(*
:Author: 

	Takashi Ichihashi Beckhoff Automation co. ltd.
	
:Date:

	2023-03-09
	
Overview
==================



Infosys Link:  `https://infosys.beckhoff.com/content/1033/tf6420_tc3_database_server/8117583755.html?id=5199556541044360835 <https://infosys.beckhoff.com/content/1033/tf6420_tc3_database_server/8117583755.html?id=5199556541044360835>`

Quick start
======================

As first you have to deine data model that the sampling data to insert to influxDB measurement.  The data models are structured by parent and child that is corresponding data tags and fields on influxDB.

.. code:: DataTag structure

	TYPE DataTag:
	STRUCT
		{attribute 'TagName' := 'machine_id'}
		machine_id : STRING(255); // 設備名
		{attribute 'TagName' := 'data_type_id'}
		data_type_id : STRING(255); // 発生イベント種別
	END_STRUCT
	END_TYPE	

	
.. code:: DataField structure

	TYPE PerformanceData EXTENDS DataTag:
	STRUCT
		{attribute 'FieldName' := 'plc_task_time'}
		task_time: UDINT;
		{attribute 'FieldName' := 'cpu_usage'}
		cpu_usage: UDINT;
		{attribute 'FieldName' := 'latency'}
		latency: UDINT;
		{attribute 'FieldName' := 'max_latency'}
		max_latency: UDINT;
		{attribute 'FieldName' := 'exceed_counter'}
		exceed_counter: UDINT;
		{attribute 'FieldName' := 'ec_lost_frames'}
		ec_lost_frames: UDINT;
		{attribute 'FieldName' := 'ec_frame_rate'}
		ec_frame_rate: LREAL;
		{attribute 'FieldName' := 'ec_lost_q_frame'}
		ec_lost_q_frames: UDINT;
		{attribute 'FieldName' := 'ec_q_frame_rate'}
		ec_q_frame_rate: LREAL;
		{attribute 'FieldName' := 'executing'}
		executing: BOOL;
		{attribute 'FieldName' := 'DB_queue_count'}
		db_insert_queue_count: UDINT;
		{attribute 'FieldName' := 'DB_buffer_current_index'}
		current_index: UDINT;
		{attribute 'FieldName' := 'DB_buffer_next_index'}
		next_index: UDINT;
	
	END_STRUCT
	END_TYPE
	
*)

FUNCTION_BLOCK RecordSQL IMPLEMENTS IRecordDB
VAR_INPUT
	nDBID						: UDINT;					// Database ID for TF6420
	DB_Parameter				: Tc2_Utilities.T_Arg;
END_VAR
VAR_OUTPUT
	bBusy			: BOOL;	// In writing database
	bError			: BOOL; // Somthing wrong situation happend
	TcResult		: Tc3_Database.I_TcMessage; // Response message
    sErrorMessage	: STRING(255);	// Error message
END_VAR
VAR
	
	//for generating timestamp
	fbGetSystemTime1: GetSystemTime;
	dwTimeLoDW: DWORD;
	dwTimeHiDW: DWORD;
	tFileTime: T_FILETIME;
	nTimestamp: LINT;
	
	//for insert samples
	fbPLCDBCmd: FB_PLCDBCmdEvt(sNetID := '', tTimeout := T#19S);
	_query								: STRING(512);
	
	// Variables for queue feature
	get_data_t 			: T_Arg;
	get_data 			: DbInsertCommand;
	State				: E_DbLogState;
END_VAR

VAR_IN_OUT
	command_queue		: CommandQueueMember;
END_VAR

CASE State OF

	E_DbLogState.idle:
		
		IF NOT fbPLCDBCmd.bBusy THEN
			State := E_DbLogState.init;
		END_IF

	E_DbLogState.init:
	
		IF NOT fbPLCDBCmd.bBusy AND command_queue.controller.num_of_data > 0 THEN
			// getting data
			get_data_t := command_queue.controller.get();
			MEMCPY(ADR(get_data), get_data_t.pData, get_data_t.cbLen);
			IF __ISVALIDREF( get_data.ref_data_buffer_counter) THEN
				get_data.ref_data_buffer_counter := get_data.ref_data_buffer_counter - get_data.chunk_size;
			END_IF
			State := E_DbLogState.writing;
		
		END_IF

	E_DbLogState.writing:
		//Write buffer element to database
		IF fbPLCDBCmd.Execute(nDBID, 
							ADR(_query), 
							SIZEOF(_query), 
							get_data.data_body.pData, 
							get_data.data_body.cbLen * get_data.chunk_size, 
							DB_Parameter.pData, 
							DB_Parameter.cbLen) THEN
			IF fbPLCDBCmd.bError THEN
				State := E_DbLogState.error;
			ELSE
				State := E_DbLogState.init;
			END_IF				
		END_IF
		

	E_DbLogState.error:
		//IF TcResult.RequestEventText(1033, sErrorMessage, SIZEOF(sErrorMessage)) THEN
            //TcResult.Send(F_GetSystemTime());
            State := E_DbLogState.idle;
            bError := TRUE;
        //END_IF

END_CASE

PROPERTY query : STRING(512)
GET
END_GET
SET
_query := query;
END_SET
END_PROPERTY

END_FUNCTION_BLOCK

(* stored: Version 1.1.0.1, ProductVersion 3.1.4024.12
   POU RecordSQL: Id {c22ca813-56d1-45d3-a2ad-9ac2c556a6da}, SpecialFunc None
   Property query: Id {c27af420-79a3-4c17-9de5-9795776e9055}
   Get Get: Id {651a9235-26b1-4e78-a03a-bd56be9eaa4a}
   Set Set: Id {57239635-62be-4167-b083-03e5cdbcae9c} *)
